TYPE DUT2 :
STRUCT
	i : INT;
	j : REAL;
	b : BOOL;
END_STRUCT
END_TYPE

(* stored: Version 1.1.0.1, ProductVersion 3.1.4024.12
   DUT DUT2: Id {6dd82a6a-193e-4588-b0de-8f1d85635ae2} *)
